{attribute 'GeneratedUsingTerminal: EL6201-0000-0017'}
{attribute addProperty BoxType "EL6201-0000-0017"}
{attribute addProperty Id "Slave_13A_DI0BOOL1Slave_13A_DI1BOOL1Slave_13A_DI2BOOL1Slave_13A_DI3BOOL1Slave_13B_DI0BOOL1Slave_13B_DI1BOOL1Slave_13B_DI2BOOL1Slave_13B_DI3BOOL1"}
{attribute addProperty CRC "1905315316"}
{attribute addProperty Size "8"}
TYPE Slave_13_Inputs_7190CDF4 :
STRUCT
	{attribute addProperty Name "Slave_13A_DI0"}
	Slave_13A_DI0 : BOOL;
	{attribute addProperty Name "Slave_13A_DI1"}
	Slave_13A_DI1 : BOOL;
	{attribute addProperty Name "Slave_13A_DI2"}
	Slave_13A_DI2 : BOOL;
	{attribute addProperty Name "Slave_13A_DI3"}
	Slave_13A_DI3 : BOOL;
	{attribute addProperty Name "Slave_13B_DI0"}
	Slave_13B_DI0 : BOOL;
	{attribute addProperty Name "Slave_13B_DI1"}
	Slave_13B_DI1 : BOOL;
	{attribute addProperty Name "Slave_13B_DI2"}
	Slave_13B_DI2 : BOOL;
	{attribute addProperty Name "Slave_13B_DI3"}
	Slave_13B_DI3 : BOOL;
END_STRUCT
END_TYPE

(* stored: Version 1.2.0.0, ProductVersion 3.1.4024.9
   DUT Slave_13_Inputs_7190CDF4: Id {5bdfb08b-c786-467a-af97-99ba99f8393a} *)
